{attribute 'GeneratedUsingTerminal: EK1122-0000-0018'}
{attribute addProperty BoxType "EK1122-0000-0018"}
{attribute addProperty Id "Beckhoff_EL3xxxsub_EK1100EK1100_AB5A94672"}
{attribute addProperty CRC "826481155"}
{attribute addProperty Size "2"}
TYPE Beckhoff_EL3xxxEK1122_31431A03 EXTENDS EK1122_AB5A9467 :
STRUCT
	{attribute addProperty Name "Beckhoff_EL3xxxsub_EK1100"}
	{attribute addProperty PreviousPort "Beckhoff EL3xxxEK1122 : D"}
	Beckhoff_EL3xxxsub_EK1100 : EK1100_AB5A9467;
END_STRUCT
END_TYPE

(* stored: Version 1.2.0.0, ProductVersion 3.1.4024.9
   DUT Beckhoff_EL3xxxEK1122_31431A03: Id {c3807f61-3138-4a2b-9a03-9b6200e6660a} *)
